{attribute 'linkalways'} 
{attribute 'no_explicit_call' := 'This FB is a CLASS and must be accessed using methods or properties'}
{attribute 'enable_dynamic_creation'}
FUNCTION_BLOCK _ETcVnLineType EXTENDS EnumDatatypeBase
VAR
	localData : ETcVnLineType;
	activeData : REFERENCE TO ETcVnLineType;
	enumBaseDatatype : _DINT(localData);
END_VAR

METHOD PRIVATE AddLocalEnumeration
VAR_INPUT
	Enumeration : T_MAXSTRING;
	Value : ETcVnLineType;
END_VAR
AddEnumeration(Enumeration, Value);
END_METHOD

PROPERTY PUBLIC Address : PVOID
GET
Address := ADR(activeData);
END_GET
END_PROPERTY

METHOD PUBLIC ClearReference
VAR_INPUT
END_VAR
activeData REF= localData;
SetBaseDatatypeReference();
END_METHOD

METHOD PUBLIC Clone : I_Datatype
VAR
    pClone : POINTER TO _ETcVnLineType;
END_VAR
pClone := __NEW(_ETcVnLineType(InitialValue := Value));
Clone := pClone^;
END_METHOD

METHOD FB_init : BOOL
VAR_INPUT
	bInitRetains : BOOL; // if TRUE, the retain variables are initialized (warm start / cold start)
	bInCopyCode : BOOL;  // if TRUE, the instance afterwards gets moved into the copy code (online change)
	InitialValue : ETcVnLineType;
END_VAR
localData := InitialValue;
AddBaseDatatype(enumBaseDatatype);
ClearReference();

AddLocalEnumeration('TCVN_LT_4_CONNECTED', ETcVnLineType.TCVN_LT_4_CONNECTED);
AddLocalEnumeration('TCVN_LT_8_CONNECTED', ETcVnLineType.TCVN_LT_8_CONNECTED);
AddLocalEnumeration('TCVN_LT_ANTIALIASED', ETcVnLineType.TCVN_LT_ANTIALIASED);
END_METHOD

PROPERTY PUBLIC Identifier : T_MAXSTRING
GET
Identifier := 'ETcVnLineType';
END_GET
END_PROPERTY

METHOD IsEnumeratorValueEqual : BOOL
VAR_INPUT
	Enumerator : I_KeyValueForwardEnumerator;
END_VAR
VAR
	storedValue : ETcVnLineType;
END_VAR
IF NOT Enumerator.TryGet(storedValue) THEN
	RETURN;
END_IF

IsEnumeratorValueEqual := storedValue = activeData;
END_METHOD

METHOD PUBLIC MakeReferenceTo
VAR_INPUT
	ReferenceTarget : REFERENCE TO ETcVnLineType;
END_VAR
activeData REF= ReferenceTarget;
SetBaseDatatypeReference();
END_METHOD

METHOD PROTECTED SetBaseDatatypeReference
VAR_INPUT
END_VAR
enumBaseDatatype.MakeReferenceTo(activeData);
END_METHOD

PROPERTY PUBLIC Size : UDINT
GET
Size := SIZEOF(activeData);
END_GET
END_PROPERTY

METHOD TryMakeReferenceTo : BOOL
VAR_INPUT
	Target : I_Datatype;
END_VAR
VAR
	targetAsEnum : I_EnumDatatype;
	pTargetData : POINTER TO ETcVnLineType;
END_VAR
IF NOT Target.TryResolveAsEnumDatatype(targetAsEnum) THEN
	RETURN;
END_IF

IF targetAsEnum.Identifier <> Identifier THEN
	RETURN;
END_IF

pTargetData := Target.Address;
activeData REF= pTargetData^;
SetBaseDatatypeReference();
TryMakeReferenceTo := TRUE;
END_METHOD

PROPERTY PUBLIC Value : ETcVnLineType
GET
Value := activeData;
END_GET
SET
activeData := Value;
END_SET
END_PROPERTY

END_FUNCTION_BLOCK

(* stored: Version 1.1.0.1
   POU _ETcVnLineType: Id {82230840-5104-418c-a98d-0726d7c220ac}, SpecialFunc None
   Folder Constructor: Id {48ff096b-c4be-43f7-b3d6-35b9e3528c3f}
   Folder Private: Id {d870258c-eb3c-4679-9385-d881b875fb88}
   Folder Protected: Id {edac36a5-6e29-4c4e-9236-5241c53bf188}
   Method AddLocalEnumeration: Id {4954d175-45f0-498b-9e4c-c8c3c0e3cf17}
   Property Address: Id {5285637a-b73d-4fb3-b7b8-aafed831e2d3}
   Get Get: Id {61d75fff-0c50-442d-a9af-d55b4f558d13}
   Method ClearReference: Id {c8138ba2-491f-48f3-9d55-13933049023d}
   Method Clone: Id {e367fe98-5ee3-4822-9518-2f8930e16523}
   Method FB_init: Id {9dcd3986-a674-411e-85c4-6b911d73fe09}
   Property Identifier: Id {3ed34665-041d-439d-bd41-7adc95043124}
   Get Get: Id {0d47ec52-383d-40f4-b0ba-e6780f06b17f}
   Method IsEnumeratorValueEqual: Id {944af466-5c2b-4428-b23a-2003afa766d9}
   Method MakeReferenceTo: Id {4ce91b92-21b1-45a1-88e2-fc6c8c077ea4}
   Method SetBaseDatatypeReference: Id {e4695c86-2323-4444-bba8-9796f13c7c05}
   Property Size: Id {898e536f-dc84-4e09-b682-bb037d6f7685}
   Get Get: Id {8c3cfbea-efaf-4d29-9933-25b8338fa976}
   Method TryMakeReferenceTo: Id {7787ca07-8906-416c-9abb-3cb56a3f3963}
   Property Value: Id {11af1d05-876a-4a79-a861-8e430594d637}
   Get Get: Id {7096c7c7-924f-4fea-bff9-ae27730d77de}
   Set Set: Id {61ab1500-a95c-405e-b85d-1ac0b0778b83} *)
